(* CODESYS project WagoLibPythonExternal_v0.0.1.library
   DefaultNamespace: WagoLibPythonExternalFile
   Author: Jesse Cox - USA
   Title: WagoLibPythonExternalFile
   Version: 0.0.1
   Description: This library allows a program to use python scripts added as external files.
   Company: WAGO Corp. USA

Project tree, tasks and I/O mapping:
  libraries: ; SysProcess, 3.5.7.0 (System); ISysTypes2, 3.5.0.0 (System)
  00000000-0000-0000-0000-000000000000|C:\Users\Jesse\Desktop\EcPyTest.py
  function block fbPythonCall [ST]
*)

// fbPythonCall
FUNCTION_BLOCK fbPythonCall
VAR_IN_OUT
	xExecute	: BOOL;
	asArgv		: ARRAY[*] OF STRING;
END_VAR
VAR_INPUT
	sFileName	: STRING(80);
END_VAR
VAR_OUTPUT
	sReturnData	: STRING(255);
END_VAR
VAR
	sShellString	: STRING(255);
	ub: DINT;
	lb: DINT;
	i: DINT;
	diShellReturn: DINT := 255;
	udiShellNumOfChars: UDINT := 255;
	typShellRslt: RTS_IEC_RESULT;
	xStringBuilt: BOOL;
END_VAR

ub:=UPPER_BOUND (asArgv,1);
lb:=LOWER_BOUND (asArgv,1);

IF xExecute THEN
	IF NOT xStringBuilt THEN
	sShellString := CONCAT('python /home/codesys_root/PlcLogic/Application/', sFileName);
		FOR i := lb TO ub DO
			sShellString := CONCAT(sShellString, ' ');
			sShellString := CONCAT(sShellString, asArgv[i]);
			IF i = ub THEN
				xStringBuilt := TRUE;
			END_IF
		END_FOR
	END_IF
	diShellReturn := SysProcess.SysProcessExecuteCommand2(	pszCommand:= sShellString, 
															pszStdOut:= sReturnData, 
															udiStdOutLen:= udiShellNumOfChars, 
															pResult:= typShellRslt);
	IF diShellReturn > 1 THEN
		xStringBuilt := FALSE;
		diShellReturn := 0;
		xExecute := FALSE;
	END_IF	
END_IF

END_FUNCTION_BLOCK
